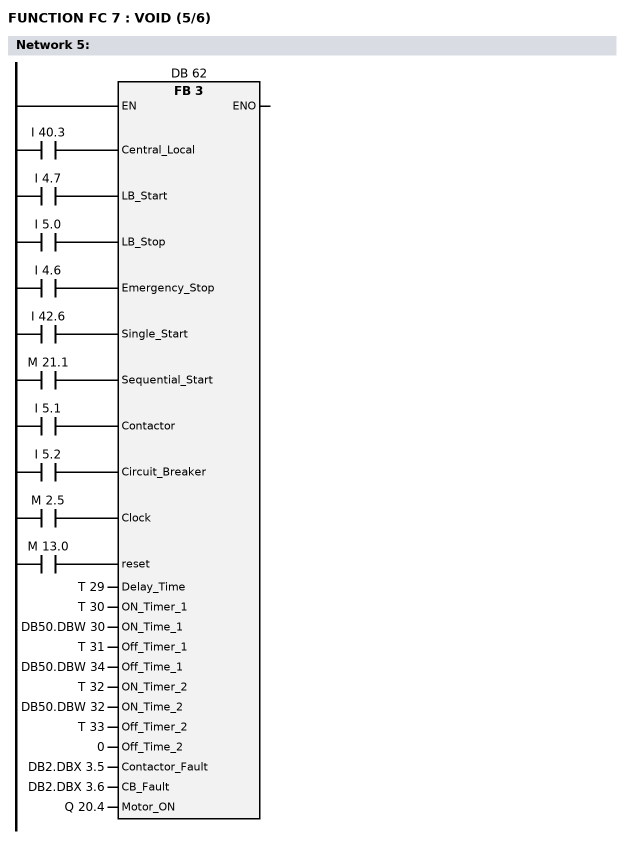

      A     I     40.3;
      =     L      0.0;
      BLD   103;
      A     I      4.7;
      =     L      0.1;
      BLD   103;
      A     I      5.0;
      =     L      0.2;
      BLD   103;
      A     I      4.6;
      =     L      0.3;
      BLD   103;
      A     I     42.6;
      =     L      0.4;
      BLD   103;
      A     M     21.1;
      =     L      0.5;
      BLD   103;
      A     I      5.1;
      =     L      0.6;
      BLD   103;
      A     I      5.2;
      =     L      0.7;
      BLD   103;
      A     M      2.5;
      =     L      1.0;
      BLD   103;
      A     M     13.0;
      =     L      1.1;
      BLD   103;
      CALL FB     3 , DB    62 (
           Central_Local            := L      0.0,
           LB_Start                 := L      0.1,
           LB_Stop                  := L      0.2,
           Emergency_Stop           := L      0.3,
           Single_Start             := L      0.4,
           Sequential_Start         := L      0.5,
           Contactor                := L      0.6,
           Circuit_Breaker          := L      0.7,
           Clock                    := L      1.0,
           reset                    := L      1.1,
           Delay_Time               := T     29,
           ON_Timer_1               := T     30,
           ON_Time_1                := DB50.DBW   30,
           Off_Timer_1              := T     31,
           Off_Time_1               := DB50.DBW   34,
           ON_Timer_2               := T     32,
           ON_Time_2                := DB50.DBW   32,
           Off_Timer_2              := T     33,
           Off_Time_2               := 0,
           Contactor_Fault          := DB2.DBX    3.5,
           CB_Fault                 := DB2.DBX    3.6,
           Motor_ON                 := Q     20.4);
      NOP   0;
NETWORK
TITLE =
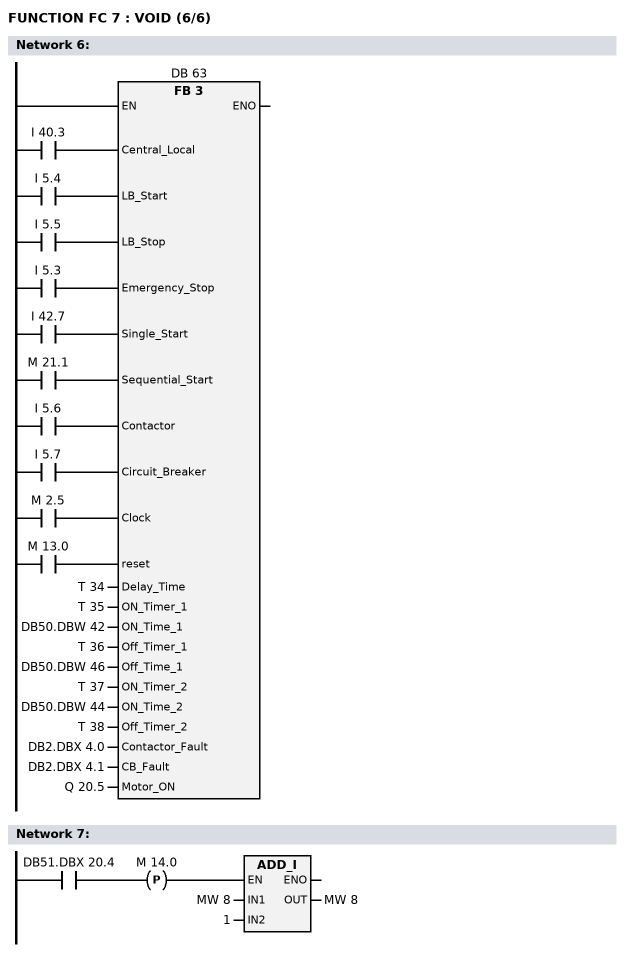

      A     I     40.3;
      =     L      0.0;
      BLD   103;
      A     I      5.4;
      =     L      0.1;
      BLD   103;
      A     I      5.5;
      =     L      0.2;
      BLD   103;
      A     I      5.3;
      =     L      0.3;
      BLD   103;
      A     I     42.7;
      =     L      0.4;
      BLD   103;
      A     M     21.1;
      =     L      0.5;
      BLD   103;
      A     I      5.6;
      =     L      0.6;
      BLD   103;
      A     I      5.7;
      =     L      0.7;
      BLD   103;
      A     M      2.5;
      =     L      1.0;
      BLD   103;
      A     M     13.0;
      =     L      1.1;
      BLD   103;
      CALL FB     3 , DB    63 (
           Central_Local            := L      0.0,
           LB_Start                 := L      0.1,
           LB_Stop                  := L      0.2,
           Emergency_Stop           := L      0.3,
           Single_Start             := L      0.4,
           Sequential_Start         := L      0.5,
           Contactor                := L      0.6,
           Circuit_Breaker          := L      0.7,
           Clock                    := L      1.0,
           reset                    := L      1.1,
           Delay_Time               := T     34,
           ON_Timer_1               := T     35,
           ON_Time_1                := DB50.DBW   42,
           Off_Timer_1              := T     36,
           Off_Time_1               := DB50.DBW   46,
           ON_Timer_2               := T     37,
           ON_Time_2                := DB50.DBW   44,
           Off_Timer_2              := T     38,
           Contactor_Fault          := DB2.DBX    4.0,
           CB_Fault                 := DB2.DBX    4.1,
           Motor_ON                 := Q     20.5);
      NOP   0;
NETWORK
TITLE =

      A     DB51.DBX   20.4;
      FP    M     14.0;
      JNB   _001;
      L     MW     8;
      L     1;
      +I    ;
      T     MW     8;
_001: NOP   0;
END_FUNCTION

ORGANIZATION_BLOCK OB 1
TITLE = "Main Program Sweep (Cycle)"
VERSION : 0.1


VAR_TEMP
  OB1_EV_CLASS : BYTE ;	//Bits 0-3 = 1 (Coming event), Bits 4-7 = 1 (Event class 1)
  OB1_SCAN_1 : BYTE ;	//1 (Cold restart scan 1 of OB 1), 3 (Scan 2-n of OB 1)
  OB1_PRIORITY : BYTE ;	//Priority of OB Execution
  OB1_OB_NUMBR : BYTE ;	//1 (Organization block 1, OB1)
  OB1_RESERVED_1 : BYTE ;	//Reserved for system
  OB1_RESERVED_2 : BYTE ;	//Reserved for system
  OB1_PREV_CYCLE : INT ;	//Cycle time of previous OB1 scan (milliseconds)
  OB1_MIN_CYCLE : INT ;	//Minimum cycle time of OB1 (milliseconds)
  OB1_MAX_CYCLE : INT ;	//Maximum cycle time of OB1 (milliseconds)
  OB1_DATE_TIME : DATE_AND_TIME ;	//Date and time OB1 started
END_VAR
BEGIN
NETWORK
TITLE =

      CALL FC     4 ;
      NOP   0;
NETWORK
TITLE =

      CALL FC     1 ;
      NOP   0;
NETWORK
TITLE =

      CALL FC     2 ;
      NOP   0;
NETWORK
TITLE =

      CALL FC     3 ;
      NOP   0;
NETWORK
TITLE =

      CALL FC     5 ;
      NOP   0;
NETWORK
TITLE =

      CALL FC     7 ;
      NOP   0;
NETWORK
TITLE =

      CALL FB     4 , DB    50 ;
      NOP   0;
END_ORGANIZATION_BLOCK

ORGANIZATION_BLOCK OB 82
VERSION : 0.1


VAR_TEMP
  TEMP0 : BYTE ;
  TEMP1 : BYTE ;
  TEMP2 : BYTE ;
  TEMP3 : BYTE ;
  TEMP4 : BYTE ;
  TEMP5 : BYTE ;
  TEMP6 : WORD ;
  TEMP7 : BOOL ;
  TEMP8 : BOOL ;
  TEMP9 : BOOL ;
  TEMP10 : BOOL ;
  TEMP11 : BOOL ;
  TEMP12 : BOOL ;
  TEMP13 : BOOL ;
  TEMP14 : BOOL ;
  TEMP15 : BYTE ;
  TEMP16 : BOOL ;
  TEMP17 : BOOL ;
  TEMP18 : BOOL ;
  TEMP19 : BOOL ;
  TEMP20 : BOOL ;
  TEMP21 : BOOL ;
  TEMP22 : BOOL ;
  TEMP23 : BOOL ;
  TEMP24 : BOOL ;
  TEMP25 : BOOL ;
  TEMP26 : BOOL ;
  TEMP27 : BOOL ;
  TEMP28 : BOOL ;
  TEMP29 : BOOL ;
  TEMP30 : BOOL ;
  TEMP31 : BOOL ;
  TEMP32 : DATE_AND_TIME ;
END_VAR
BEGIN
END_ORGANIZATION_BLOCK

ORGANIZATION_BLOCK OB 85
TITLE = "Organization Block (OB) Not Loaded Fault"
VERSION : 0.1


VAR_TEMP
  OB85_EV_CLASS : BYTE ;	//16#35 Event class 3
  OB85_FLT_ID : BYTE ;	//16#XX, Fault identification code
  OB85_PRIORITY : BYTE ;	//Priority of OB Execution
  OB85_OB_NUMBR : BYTE ;	//85 (Organization block 85, OB85)
  OB85_RESERVED_1 : BYTE ;	//Reserved for system
  OB85_RESERVED_2 : BYTE ;	//Reserved for system
  OB85_RESERVED_3 : INT ;	//Reserved for system
  OB85_ERR_EV_CLASS : BYTE ;	//Class of event causing error
  OB85_ERR_EV_NUM : BYTE ;	//Number of event causing error
  OB85_OB_PRIOR : BYTE ;	//Priority of OB causing error
  OB85_OB_NUM : BYTE ;	//Number of OB causing error
  OB85_DATE_TIME : DATE_AND_TIME ;	//Date and time OB85 started
END_VAR
BEGIN
END_ORGANIZATION_BLOCK

ORGANIZATION_BLOCK OB 86
VERSION : 0.1


VAR_TEMP
  TEMP0 : BYTE ;
  TEMP1 : BYTE ;
  TEMP2 : BYTE ;
  TEMP3 : BYTE ;
  TEMP4 : BYTE ;
  TEMP5 : BYTE ;
  TEMP6 : WORD ;
  //TEMP7 : ARRAY  [0 .. 31 ] OF BOOL ;
  TEMP8 : DATE_AND_TIME ;
END_VAR
BEGIN
END_ORGANIZATION_BLOCK

ORGANIZATION_BLOCK OB 87
TITLE = "Communication Fault"
VERSION : 0.1


VAR_TEMP
  OB87_EV_CLASS : BYTE ;	//16#39 Event class 3
  OB87_FLT_ID : BYTE ;	//16#XX, Fault identifcation code
  OB87_PRIORITY : BYTE ;	//Priority of OB Execution
  OB87_OB_NUMBR : BYTE ;	//87 (Organization block 87, OB87)
  OB87_RESERVED_1 : BYTE ;	//Reserved for system
  OB87_RESERVED_2 : BYTE ;	//Reserved for system
  OB87_RESERVED_3 : WORD ;	//Reserved for system
  OB87_RESERVED_4 : DWORD ;	//Reserved for system
  OB87_DATE_TIME : DATE_AND_TIME ;	//Date and time OB87 started
END_VAR
BEGIN
END_ORGANIZATION_BLOCK

ORGANIZATION_BLOCK OB 121
TITLE = "Programming Error"
VERSION : 0.1


VAR_TEMP
  OB121_EV_CLASS : BYTE ;	//16#25, Event class 2, Entering event state, Internal fault event
  OB121_SW_FLT : BYTE ;	//16#XX Software programming fault
  OB121_PRIORITY : BYTE ;	//Priority of OB Execution
  OB121_OB_NUMBR : BYTE ;	//121 (Organization block 121, OB121)
  OB121_BLK_TYPE : BYTE ;	//16#88/8A/8B/8C/8E Type of block fault occured in
  OB121_RESERVED_1 : BYTE ;	//Reserved for system
  OB121_FLT_REG : WORD ;	//16#XX Specific register that caused fault
  OB121_BLK_NUM : WORD ;	//Number of block that programming fault occured in
  OB121_PRG_ADDR : WORD ;	//Address in block where programming fault occured
  OB121_DATE_TIME : DATE_AND_TIME ;	//Date and time OB121 started
END_VAR
BEGIN
END_ORGANIZATION_BLOCK

ORGANIZATION_BLOCK OB 122
VERSION : 0.1


VAR_TEMP
  TEMP0 : BYTE ;
  TEMP1 : BYTE ;
  TEMP2 : BYTE ;
  TEMP3 : BYTE ;
  TEMP4 : BYTE ;
  TEMP5 : BYTE ;
  TEMP6 : WORD ;
  TEMP7 : WORD ;
  TEMP8 : WORD ;
  TEMP9 : DATE_AND_TIME ;
END_VAR
BEGIN
END_ORGANIZATION_BLOCK

